VAR_GLOBAL CONSTANT
    gc_iSizeOfGGOArray : INT := 50;
    gc_GaugeValidState :	INT := 4;
END_VAR

(* stored: Version 1.1.0.1, ProductVersion 3.1.4022.18
   GVL Constants: Id {352ad9bf-a34d-4366-bd0d-dad0c46d83d9} *)
